{attribute 'GeneratedUsingTerminal: EK1100-0000-0018'}
{attribute addProperty BoxType "EK1100-0000-0018"}
{attribute addProperty Id "Beckhoff_EPP9xxxEK1122Beckhoff_EPP9xxxEK1122_03A068BC102"}
{attribute addProperty CRC "4168416555"}
{attribute addProperty Size "102"}
TYPE Beckhoff_EPP9xxx_F874FD2B EXTENDS EK1100_AB5A9467 :
STRUCT
	{attribute addProperty Name "Beckhoff_EPP9xxxEK1122"}
	Beckhoff_EPP9xxxEK1122 : Beckhoff_EPP9xxxEK1122_03A068BC;
END_STRUCT
END_TYPE

(* stored: Version 1.2.0.0, ProductVersion 3.1.4024.9
   DUT Beckhoff_EPP9xxx_F874FD2B: Id {b167d3db-3e81-46fd-aa6b-92a9d45c5138} *)
